PROGRAM S_Master_SMAC
VAR	 
eState								: E_SmacState;
	
/////////////////////////////////////////////INITIALIZATION FUNCTION/////////////////////////////////////////////////////
	fbSmacInitialization_L							: FB_SmacInitialization;
	I_O_fbSmacInitialization_L						:ST_Phasing_Home;

	fbSmacInitialization_R							: FB_SmacInitialization;
	I_O_fbSmacInitialization_R						:ST_Phasing_Home;

/////////////////////////////////////////////CYCLE/MANUAL FUNCTION/////////////////////////////////////////////////////
	fbSmacCycleMan									: FB_SmacCycleMan;
	bTest											: BOOL;
/////////////////////////////////////////////CTRL SMAC/////////////////////////////////////////////////////
	nHomeState										: DINT;	
	nCyclePickState									: DINT;
	nCycleScrewkState								: DINT;
	nHomeStateManual								: DINT;	
	nCyclePickStateManual							: DINT;
	nCycleScrewkStateManual							: DINT;
	bLinealHomed									: BOOL;
	bRotativeHomed									: BOOL;
	bFirstCycle										: BOOL;
	
	
	aCycleFlag										: ARRAY[0..10] OF BOOL;

/////////////////////////////////////////////ERROR FUNCTION/////////////////////////////////////////////////////	
	fbErrorRST										: FB_ErrorReset;
	bEnbale_ErrorRST								: BOOL;
	bResetErrors									: BOOL;
	bAllErrorsCleared								: BOOL;
/////////////////////////////////////////////TIMERS / TRIGGERS/////////////////////////////////////////////////////
	tonResetError									:Tc2_Standard.TON;
	tonAbortModule									:Tc2_Standard.TON;
	tonCaseDelay									: ARRAY[0..40] OF TON;
	rTrigCase										: ARRAY[0..10] OF R_TRIG;
	CMDTrig											: ARRAY[0..10] OF R_TRIG;										
/////////////////////////////////////////////GRIPPERS CONTROL/////////////////////////////////////////////////////
	bCatchPiece							:BOOL;	//If set to TRUE - gripper OPEN || FALSE - gripper CLOSED
	bGuideScrew							:BOOL;	//If set to TRUE - gripper OPEN || FALSE - gripper CLOSED
	bGripperGuide_Timeout				:BOOL;	//Gripper didn't close in 3sec
	bGripperFixture_Timeout				:BOOL;	//Gripper didn't close in 3sec
	fbGripper_Guide						:FB_GripperCtrl;	
	fbGripper_Fixture					:FB_GripperCtrl;

END_VAR//---------------------------------------------------------------------------------------oldschoo1
VAR_OUTPUT
	stSmacReport						:ST_ProcessReport;
END_VAR

//--------------------IN/OUT----------------------------------------*
VAR_INPUT
	bCloseGripper						: BOOL;
	CMD									:ST_ModuleCMD;	
END_VAR
VAR_OUTPUT
	STATUS								:ST_ModuleStatus;
	I_O_fbSmacCycleMan					: ST_CYC_MAN;
END_VAR




//----------------------------------------------------------oldschoo1

PRG_Fault_SMAC(aAlarms := GVL_Master.stAlarms);
b_Ctrl_Smac();
c_FunctionProcess();
d_TimTrig();

ACTION a_StringDefinitions:

//////////////////////////////////////////STATUS STRING DEFINITIONS/////////////////////////////////////////////////////

	stSmacIO.sStatus[0]:='Initialization done';
	stSmacIO.sStatus[1]:='Servo enabled';
	stSmacIO.sStatus[2]:='';
	stSmacIO.sStatus[3]:='Motion execution acknowledge bit';
	stSmacIO.sStatus[4]:='Trajectory complete';
	stSmacIO.sStatus[5]:='';
	stSmacIO.sStatus[6]:='Homing Success';
	stSmacIO.sStatus[7]:='Homing failure';
	stSmacIO.sStatus[8]:='Phasing Succes';
	stSmacIO.sStatus[9]:='Phasing failure';
	stSmacIO.sStatus[10]:='Macro execution error';
	stSmacIO.sStatus[11]:='Macro execution';
	stSmacIO.sStatus[12]:='General fault';
	stSmacIO.sStatus[13]:='Servo error';
	stSmacIO.sStatus[14]:='STO fault';
	stSmacIO.sStatus[15]:='STO status';
	stSmacIO.sStatus[16]:='STO Input 1 de-energized';
	stSmacIO.sStatus[17]:='STO Input 2 de-energized';
	stSmacIO.sStatus[18]:='I2T fault';
	stSmacIO.sStatus[19]:='Driver overtemperature fault';
	stSmacIO.sStatus[20]:='Initialization done';
	
//////////////////////////////////////////MODE OF OPERATION STRING DEFINITIONS/////////////////////////////////////////////////////
	
	stSmacIO.sModeOfOperation[0] :='';
	stSmacIO.sModeOfOperation[1] :='Absolute position move';
	stSmacIO.sModeOfOperation[2] :='Relative position move';
	stSmacIO.sModeOfOperation[3] :='Velocity move';
	stSmacIO.sModeOfOperation[4] :='Torque move';
	stSmacIO.sModeOfOperation[5] :='Current move/QM1';
	stSmacIO.sModeOfOperation[6] :='Homing';
	stSmacIO.sModeOfOperation[7] :='Phasing';
	stSmacIO.sModeOfOperation[8] :='Current move/QM2';
	stSmacIO.sModeOfOperation[9] :='';
	stSmacIO.sModeOfOperation[10] :='Macro execution**';
	
//////////////////////////////////////////CONTRO WORD STRING DEFINITIONS/////////////////////////////////////////////////////

stSmacIO.sControlWord[0] :='';
stSmacIO.sControlWord[1] :='Start motion/macro start';
stSmacIO.sControlWord[2] :='Stop motion';
stSmacIO.sControlWord[3] :='Motor off';
stSmacIO.sControlWord[4] :='Motor on';
stSmacIO.sControlWord[5] :='Fault reset';
END_ACTION

ACTION b_Ctrl_Smac:

IF cmd.bAbort OR NOT stSafety.bSafety_OK OR NOT cmd.bEnable   THEN
	eState									:= E_SmacState.ABORTED;
END_IF

IF CMDTrig[4].Q THEN
	eState									:= E_SmacState.RESET_ERROR;
END_IF

IF eState = E_SmacState.MANUAL THEN
	I_O_fbSmacCycleMan.bManual_fbSmacCycleMan := TRUE;
ELSE I_O_fbSmacCycleMan.bManual_fbSmacCycleMan := FALSE;
END_IF

IF CMD.bManualMode THEN
	eState									:= E_SmacState.MANUAL;
END_IF
									

CMDTrig[0]( CLK := cmd.bAbort OR NOT stSafety.bSafety_OK OR NOT cmd.bEnable );
CMDTrig[1]( CLK := CMD.bEnable AND tonCaseDelay[3].Q );
CMDTrig[2]( CLK := CMD.bExecute);
CMDTrig[3]( CLK := CMD.bManualMode);
CMDTrig[4]( CLK := CMD.bReset);

		
(*******************************************************CTRL***********************************************************)
// Axis CTRL State Machine
CASE eState OF //--------------------------------------------------------------------------------------------------SM
	
E_SmacState.ABORTED://-------------------------------------------------------------------------------------------ABORTED:

						IF tonCaseDelay[22].Q THEN
							eState 												:= E_SmacState.ERROR;						
						END_IF

						IF  CMD.bEnable THEN
							eState 												:= E_SmacState.HOMING;
						END_IF
						//RESETTING
						I_O_fbSmacInitialization_R.bFunctionRequest				:= FALSE;
						I_O_fbSmacInitialization_L.bFunctionRequest				:= FALSE;
						I_O_fbSmacInitialization_R.bReset						:= TRUE;
						I_O_fbSmacInitialization_L.bReset						:= TRUE;
						I_O_fbSmacInitialization_L.bAcknowledge					:= FALSE;
						I_O_fbSmacInitialization_R.bAcknowledge					:= FALSE;
						
						I_O_fbSmacCycleMan.bAutoCycleRequest					:= FALSE;
						I_O_fbSmacCycleMan.bResetAutoCycle						:= TRUE;
						I_O_fbSmacCycleMan.bInitSecondPart						:= FALSE;
						I_O_fbSmacCycleMan.bAutoCycleAcknowledge				:= FALSE;
						aCycleFlag[1]											:= FALSE;
						aCycleFlag[2]											:= FALSE;
						aCycleFlag[3]											:= FALSE;
						
						nHomeState												:= 0;
						nCyclePickState											:= 0;
						nCycleScrewkState										:= 0;
						
						bCloseGripper											:= FALSE;
						
						IF tonCaseDelay[3].Q THEN
							I_O_fbSmacInitialization_R.bReset					:= FALSE;
							I_O_fbSmacInitialization_L.bReset					:= FALSE;
							I_O_fbSmacInitialization_R.bEnable					:= FALSE;
							I_O_fbSmacInitialization_L.bEnable					:= FALSE;
							
							I_O_fbSmacCycleMan.bResetAutoCycle					:= FALSE;
							I_O_fbSmacCycleMan.bCycProcess						:= FALSE;
							
							I_O_fbSmacCycleMan.bResetAutoCycle					:= FALSE;
							I_O_fbSmacCycleMan.bCycProcess						:= FALSE;
						END_IF
						

E_SmacState.HOMING://---------------------------------------------------------------------------------------------HOMING:
////////////////////////////////////////////////////LINEAL HOME////////////////////////////////////////////////////
						CASE 	nHomeState	OF
								
						0:
						IF aCycleFlag[1] THEN
							eState 												:= E_SmacState.AXIS_READY;
						ELSE nHomeState											:= 200;
						END_IF
						200:
						I_O_fbSmacInitialization_L.bEnable						:= TRUE;
						IF tonCaseDelay[6].Q THEN
							nHomeState											:= 300;
						END_IF
						300:
						I_O_fbSmacInitialization_L.bFunctionRequest				:= TRUE;
						IF tonCaseDelay[7].Q THEN
							nHomeState											:= 400;
						END_IF
						400:
						IF I_O_fbSmacInitialization_L.bAcknowledgeRequest THEN
							I_O_fbSmacInitialization_L.bAcknowledge				:= TRUE;
							nHomeState											:= 500;
							bLinealHomed										:= TRUE;
						ELSIF I_O_fbSmacInitialization_L.bPhasingError OR I_O_fbSmacInitialization_L.bHomeError THEN
							nHomeState											:= 500;
						END_IF
						500:
						I_O_fbSmacInitialization_L.bReset						:= TRUE;
						IF tonCaseDelay[8].Q THEN
							nHomeState											:= 600;
						END_IF
						600:
						I_O_fbSmacInitialization_L.bEnable						:= FALSE;
						I_O_fbSmacInitialization_L.bReset						:= FALSE;
						I_O_fbSmacInitialization_L.bFunctionRequest				:= FALSE;
						I_O_fbSmacInitialization_L.bAcknowledge					:= FALSE;
						IF bLinealHomed THEN
							nHomeState											:= 1200;
						END_IF
						
						1200:
						I_O_fbSmacInitialization_R.bEnable						:= TRUE;
						IF tonCaseDelay[9].Q THEN
							nHomeState											:= 1300;
						END_IF
						1300:
						I_O_fbSmacInitialization_R.bFunctionRequest				:= TRUE;
						IF tonCaseDelay[10].Q THEN
							nHomeState											:= 1400;
						END_IF
						1400:
						IF I_O_fbSmacInitialization_R.bAcknowledgeRequest THEN
							I_O_fbSmacInitialization_R.bAcknowledge				:= TRUE;
							nHomeState											:= 1500;
							bRotativeHomed										:= TRUE;
						ELSIF I_O_fbSmacInitialization_R.bPhasingError OR I_O_fbSmacInitialization_R.bHomeError THEN
							nHomeState											:= 1500;
						END_IF
						1500:
						I_O_fbSmacInitialization_R.bReset						:= TRUE;
						IF tonCaseDelay[11].Q THEN
							nHomeState											:= 1600;
						END_IF
						1600:
						I_O_fbSmacInitialization_R.bEnable						:= FALSE;
						I_O_fbSmacInitialization_R.bReset						:= FALSE;
						I_O_fbSmacInitialization_R.bFunctionRequest				:= FALSE;
						I_O_fbSmacInitialization_R.bAcknowledge					:= FALSE;
						IF bRotativeHomed AND bLinealHomed THEN
							bRotativeHomed										:= FALSE;
							bLinealHomed										:= FALSE;
							aCycleFlag[1]										:= TRUE;
							nHomeState											:= 0;
						END_IF
						
						5000://ERROR

						IF tonCaseDelay[12].Q THEN
							eState 												:= E_SmacState.ABORTED;
						END_IF
						END_CASE
	
						IF I_O_fbSmacInitialization_R.bHomeError OR I_O_fbSmacInitialization_R.bPhasingError OR
							I_O_fbSmacInitialization_L.bHomeError OR I_O_fbSmacInitialization_L.bPhasingError OR CMDTrig[0].Q THEN
							nHomeState											:= 5000;
						END_IF

		
E_SmacState.AXIS_READY://-------------------------------------------------------------------------------------AXIS_READY:
							
							aCycleFlag[1]										:= FALSE;
							aCycleFlag[3]										:= FALSE;
							//GO TO FIRST PART OF THE CYCLE
							IF (CMDTrig[2].Q AND stSmac.bSet_PickScrew) OR rTrigCase[1].Q THEN
									eState := E_SmacState.Cycle_Pick_Part;
							END_IF
										
							
E_SmacState.Cycle_Pick_Part://---------------------------------------------------------------------------Cycle_Pick_Part:		
							CASE nCyclePickState OF
							0:
							IF aCycleFlag[2] THEN
							eState 												:= E_SmacState.Cycle_Screw;
							ELSE nCyclePickState								:= 200;
							END_IF
							200:
							IF NOT bFirstCycle THEN
								nCyclePickState									:= 300;
							ELSE nCyclePickState								:= 400;
							END_IF
							300:
							I_O_fbSmacCycleMan.bSetValues						:= TRUE;
							IF tonCaseDelay[15].Q THEN
								nCyclePickState									:= 400;
							END_IF
							400:
							I_O_fbSmacCycleMan.bCycProcess						:= TRUE;
							IF tonCaseDelay[16].Q THEN
								nCyclePickState									:= 500;
							END_IF
							500:
							I_O_fbSmacCycleMan.bAutoCycleRequest				:= TRUE; 
							IF tonCaseDelay[17].Q THEN
								nCyclePickState									:= 600;
							END_IF
							600:
							IF I_O_fbSmacCycleMan.bFirstPartDoneFlag THEN
								aCycleFlag[2]									:= TRUE;
								nCyclePickState									:= 0;
							END_IF
							
							5000://ERROR
							IF tonCaseDelay[18].Q THEN
								eState 											:= E_SmacState.ABORTED;
							END_IF
							END_CASE
	
							IF I_O_fbSmacCycleMan.bCycError  THEN
								nCyclePickState										:= 5000;
							END_IF

						
							
							
E_SmacState.Cycle_Screw://-----------------------------------------------------------------------------------Cycle_Screw:
							aCycleFlag[2]										:= FALSE;
							CASE nCycleScrewkState OF
							0:	
							IF aCycleFlag[3] THEN//second part request
								eState 											:= E_SmacState.RECORD_CYCLE_DATA;
							ELSE nCycleScrewkState								:= 100;
							END_IF
							100:
							IF I_O_fbSmacCycleMan.bFirstPartDoneFlag AND CMDTrig[2].Q AND stSmac.bSet_ScrewItIn THEN
								I_O_fbSmacCycleMan.bInitSecondPart				:= TRUE;
								nCycleScrewkState								:= 200;
							END_IF
							200:
							bCloseGripper									:= I_O_fbSmacCycleMan.bOpenGuideGripper;
							IF I_O_fbSmacCycleMan.bAutoCycleAcknowledgeRequest THEN
								I_O_fbSmacCycleMan.bAutoCycleAcknowledge		:= TRUE;
								nCycleScrewkState								:= 300;
								
							END_IF
							300:
							IF I_O_fbSmacCycleMan.bCycleProcessDone THEN
								nCycleScrewkState								:= 400;
								I_O_fbSmacCycleMan.bAutoCycleAcknowledge		:= FALSE;
								I_O_fbSmacCycleMan.bAutoCycleRequest			:= FALSE;
								I_O_fbSmacCycleMan.bInitSecondPart				:= FALSE;
								I_O_fbSmacCycleMan.bSetValues					:= FALSE;
								I_O_fbSmacCycleMan.bResetAutoCycle				:= TRUE;
								nCycleScrewkState								:= 400;
							END_IF 
							400:
							IF tonCaseDelay[18].Q THEN
								I_O_fbSmacCycleMan.bResetAutoCycle				:= FALSE;
								I_O_fbSmacCycleMan.bCycProcess					:= FALSE;
								nCycleScrewkState								:= 500;
							END_IF
							500:
							nCycleScrewkState									:= 0;
							aCycleFlag[3]										:= TRUE;
							
							5000://ERROR
							IF tonCaseDelay[18].Q THEN
								eState 											:= E_SmacState.ABORTED;
							END_IF
							END_CASE
	
							IF I_O_fbSmacCycleMan.bCycError THEN
								nCycleScrewkState								:= 5000;
							END_IF

E_SmacState.RECORD_CYCLE_DATA://-----------------------------------------------------------------------------RECORD_CYCLE_DATA:

							
							stSmacReport.rSmac_Settings_LinearAcc				:= I_O_fbSmacCycleMan.nScaledLinearAcc;
							stSmacReport.rSmac_Settings_LinearVel				:= I_O_fbSmacCycleMan.nScaledLinearVel;
							stSmacReport.rSmac_Settings_LinearTorque			:= I_O_fbSmacCycleMan.nScaledLinearTorque;
							stSmacReport.rSmac_Settings_RotativeAcc				:= I_O_fbSmacCycleMan.nScaledRotativeAcc;
							stSmacReport.rSmac_Settings_RotativeVel				:= I_O_fbSmacCycleMan.nScaledRotativeVel;
							
							stSmacReport.bSmac_Pass								:= I_O_fbSmacCycleMan.bPass;
							stSmacReport.bSmac_Fail								:= I_O_fbSmacCycleMan.bFail;
				
							stSmacReport.rSmac_MaxDistanceReached				:= I_O_fbSmacCycleMan.MaxDistanceReached;
							IF tonCaseDelay[13].Q THEN
								eState 											:= E_SmacState.AXIS_READY;
 							END_IF
							

E_SmacState.RESET_ERROR://-----------------------------------------------------------------------------------------------ERROR:
							IF bAllErrorsCleared AND tonCaseDelay[4].Q THEN
								bEnbale_ErrorRST								:= FALSE;
							ELSE bEnbale_ErrorRST								:= TRUE;
							END_IF
							IF bFlash1Hz AND bEnbale_ErrorRST THEN
								bResetErrors									:= TRUE;
							ELSE bResetErrors									:= FALSE;
							END_IF
							IF tonCaseDelay[5].Q AND tonCaseDelay[4].Q THEN
								eState := E_SmacState.ABORTED;
							END_IF

E_SmacState.MANUAL://---------------------------------------------------------------------------------------------------MANUAL:
							IF NOT CMD.bManualMode THEN
								eState := E_SmacState.ABORTED;
							END_IF
							
ELSE 
eState := E_AxisState.ABORTED;
END_CASE //------------------------------------------------------------------------------------------------------END_CASE

(******************************************************STATUS************************************************************)
// Module Status
status.bReady					:= eState = E_SmacState.AXIS_READY;

status.bBusy					:= 	eState = E_SmacState.Cycle_Screw	OR
				   					eState = E_SmacState.Cycle_Pick_Part OR
				   					eState = E_SmacState.HOMING;
status.bFirstPartOfCycleDone	:=	I_O_fbSmacCycleMan.bFirstPartDoneFlag;	
		   
status.bDone					:= 	eState =	E_SmacState.RECORD_CYCLE_DATA;

status.bError					:= 	I_O_fbSmacInitialization_L.bHomeError OR I_O_fbSmacInitialization_R.bHomeError OR
								I_O_fbSmacInitialization_L.bPhasingError OR I_O_fbSmacInitialization_R.bPhasingError OR
								I_O_fbSmacCycleMan.bCycError OR stSmacIO.inStatusWordRotative.13 OR stSmacIO.inStatusWordLinear.13  ;
//--------------------------------------------------GRIPPERS-------------------------------------------------------------oldschoo1

IF CMD_Smac.bFixtureGripper OR (I_O_fbSmacCycleMan.bCloseFixtureGripper AND eState = E_AxisState.MANUAL_MODE) THEN
	bCatchPiece					:= TRUE;
ELSE bCatchPiece					:= FALSE;
END_IF

IF (CMD_Smac.bGuideGripper AND NOT bCloseGripper ) OR 
	(I_O_fbSmacCycleMan.bCloseGuideGripper AND eState = E_AxisState.MANUAL_MODE)THEN
	bGuideScrew					:= TRUE;
ELSE bGuideScrew					:= FALSE;
END_IF
END_ACTION

ACTION c_FunctionProcess:
//LINEAR PHASING AND HOME
fbSmacInitialization_L(	//INPUTS:
						bEnable 				:= I_O_fbSmacInitialization_L.bEnable,
						bAcknowledge 			:= I_O_fbSmacInitialization_L.bAcknowledge,
						bReset					:= I_O_fbSmacInitialization_L.bReset,
						bFunctionRequest		:= I_O_fbSmacInitialization_L.bFunctionRequest,
						nStatusWord				:= stSmacIO.inStatusWordLinear,
						nCurrentModeOfOperation	:= stSmacIO.inModeOfOperationLinear,							
						
						//OUTPUTS	
						bFunctionEnabled		=> I_O_fbSmacInitialization_L.bFunctionEnabled,
						bPhasingProcessDone		=> I_O_fbSmacInitialization_L.bPhasingProcessDone,
						bHomingProcessDone		=> I_O_fbSmacInitialization_L.bHomingProcessDone,
						bAcknowledgeRequest		=> I_O_fbSmacInitialization_L.bAcknowledgeRequest,
						bHomeError				=> I_O_fbSmacInitialization_L.bHomeError,
						bPhasingError			=> I_O_fbSmacInitialization_L.bPhasingError,
						//IN/OUT
						nControlWord			:= stSmacIO.qnControlWordLinear,								
						nModeOfOperation		:= stSmacIO.qnModeOfOperationLinear);
						
//ROTATIVE PHASING AND HOME						
fbSmacInitialization_R(	//INPUTS:
						bEnable 				:= I_O_fbSmacInitialization_R.bEnable,
						bAcknowledge 			:= I_O_fbSmacInitialization_R.bAcknowledge,
						bReset					:= I_O_fbSmacInitialization_R.bReset,
						bFunctionRequest		:= I_O_fbSmacInitialization_R.bFunctionRequest,
						nStatusWord				:= stSmacIO.inStatusWordRotative,
						nCurrentModeOfOperation	:= stSmacIO.inModeOfOperationRotative,							
						
						//OUTPUTS	
						bFunctionEnabled		=> I_O_fbSmacInitialization_R.bFunctionEnabled,
						bPhasingProcessDone		=> I_O_fbSmacInitialization_R.bPhasingProcessDone,
						bHomingProcessDone		=> I_O_fbSmacInitialization_R.bHomingProcessDone,
						bAcknowledgeRequest		=> I_O_fbSmacInitialization_R.bAcknowledgeRequest,
						bHomeError				=> I_O_fbSmacInitialization_R.bHomeError,
						bPhasingError			=> I_O_fbSmacInitialization_R.bPhasingError,
						//IN/OUT
						nControlWord			:= stSmacIO.qnControlWordRotative,								
						nModeOfOperation		:= stSmacIO.qnModeOfOperationRotative);
//CYCLE / MANUAL						
fbSmacCycleMan(			//INPUTS:
						nLinearVel				:= I_O_fbSmacCycleMan.nLinearVel,
						nLinearAcc				:= I_O_fbSmacCycleMan.nLinearAcc,
						nLinearSetPoint			:= I_O_fbSmacCycleMan.nLinearSetPoint,
						nLinearTorque			:= I_O_fbSmacCycleMan.nLinearTorque,
						bRotativeWorkPosition	:= I_O_fbSmacCycleMan.nRotativeWorkPosition,
						
						nRotativeVel			:= I_O_fbSmacCycleMan.nRotativeVel,
						nRotativeAcc			:= I_O_fbSmacCycleMan.nRotativeAcc,
						nRotativeSetPoint		:=  GVL_PERSISTENT.nSmacRotativeSetPoint,
						
						bCycProcess				:= I_O_fbSmacCycleMan.bCycProcess,
						bAutoCycleAcknowledge	:= I_O_fbSmacCycleMan.bAutoCycleAcknowledge,
						bAutoCycleRequest		:= I_O_fbSmacCycleMan.bAutoCycleRequest,
						bResetAutoCycle			:= I_O_fbSmacCycleMan.bResetAutoCycle,
						bInitSecondPart			:= I_O_fbSmacCycleMan.bInitSecondPart,
						bSetValues				:= GVL_HMI.bSmacSetValue OR (NOT bFirstCycle AND I_O_fbSmacCycleMan.bSetValues),
						bFixtureGripperClosed	:= stSmac.bGripperB_ClosedSensor,
						bGuideGripperClosed		:= stSmac.bGripperA_ClosedSensor,
						bManual					:= I_O_fbSmacCycleMan.bManual_fbSmacCycleMan,
						
						nDistanceSetPoint		:= I_O_fbSmacCycleMan.nDistanceSetPoint,				
						nDistanceTolerance		:= 500, //I_O_fbSmacCycleMan.nDistanceTolerance,
						bPickCycleMan			:= GVL_HMI.bSmacCyc1,
						bScrewCycleMan			:= GVL_HMI.bSmacCyc2,
						bHomeMan				:= GVL_HMI.bSmacHOME,
						//OUTPUTS
						bAutoCycleAcknowledgeRequest 	=> I_O_fbSmacCycleMan.bAutoCycleAcknowledgeRequest,
						bCycleProcessDone				=> I_O_fbSmacCycleMan.bCycleProcessDone,
						bFirstPartDoneFlag				=> I_O_fbSmacCycleMan.bFirstPartDoneFlag,
						bCycError						=> I_O_fbSmacCycleMan.bCycError,
						bOpenGuideGripper				=> I_O_fbSmacCycleMan.bOpenGuideGripper,
						bCloseGuideGripper				=> I_O_fbSmacCycleMan.bCloseGuideGripper,
						bCloseFixtureGripper			=> I_O_fbSmacCycleMan.bCloseFixtureGripper,
						bPass							=> I_O_fbSmacCycleMan.bPass,										
						bFail							=> I_O_fbSmacCycleMan.bFail,
						
						nScaledLinearVel				=> I_O_fbSmacCycleMan.nScaledLinearVel,			
						nScaledLinearAcc				=> I_O_fbSmacCycleMan.nScaledLinearAcc,						
						nScaledLinearSetPoint			=> I_O_fbSmacCycleMan.nScaledLinearSetPoint,						
						nScaledLinearTorque				=> I_O_fbSmacCycleMan.nScaledLinearTorque,					
	
						nScaledRotativeVel				=> I_O_fbSmacCycleMan.nScaledRotativeVel,						
						nScaledRotativeAcc				=> I_O_fbSmacCycleMan.nScaledRotativeAcc,					
						nScaledRotativeSetPoint			=> I_O_fbSmacCycleMan.nScaledRotativeSetPoint,
						MaxDistanceReached				=> I_O_fbSmacCycleMan.MaxDistanceReached,	
						bScrewAnimation					=> GVL_HMI.bScrewAnimation,
						//IN/OUT
						stSmacIO				:= stSmacIO);
						
							
									
												
//ERROR RESET
fbErrorRST(				//INPUTS
						bEnbale					:= bEnbale_ErrorRST,
						bResetErrors			:= bResetErrors,
						//OUTPUTS
						bAllErrorsCleared		=> bAllErrorsCleared,
						//IN/OUT
						stSmacIO				:= stSmacIO,
						bHomeError_L			:= I_O_fbSmacInitialization_L.bHomeError,
						bHomeError_R			:= I_O_fbSmacInitialization_R.bHomeError,
						bPhasingError_L			:= I_O_fbSmacInitialization_L.bPhasingError,
						bPhasingError_R			:= I_O_fbSmacInitialization_R.bPhasingError,
						bCycleError				:= I_O_fbSmacCycleMan.bCycError);

// Grippers CTRL
fbGripper_Fixture	 (bCloseGrip		:=bCatchPiece,
					  bClosedSensor		:=stSmac.bGripperB_ClosedSensor,
					  bOpen_Sig			=>stSmac.bGripperB_Open,
					  bClose_Sig		=>stSmac.bGripperB_Close,
					  bTimeout			=>bGripperFixture_Timeout);


fbGripper_Guide	     (bCloseGrip		:=bGuideScrew,
					  bClosedSensor		:=stSmac.bGripperA_ClosedSensor,
					  bOpen_Sig			=>(stSmac.bGripperA_Open ),
					  bClose_Sig		=>stSmac.bGripperA_Close,
					  bTimeout			=>bGripperGuide_Timeout);
END_ACTION

ACTION d_TimTrig:
//TIMERS

tonCaseDelay[0](IN := (eState =E_SmacState.HOMING) , PT := T#1S);
tonCaseDelay[1(*10*)](IN := eState = E_SmacState.Cycle_Screw , PT := T#1S);
tonCaseDelay[16](IN := eState = E_SmacState.Cycle_Pick_Part , PT := T#500MS);
tonCaseDelay[3](IN := (eState = E_SmacState.ABORTED) , PT := T#1S);
tonCaseDelay[4](IN := eState = E_SmacState.ERROR , PT := T#1S);
tonCaseDelay[13](IN := eState = E_SmacState.RECORD_CYCLE_DATA , PT := T#500MS);


tonCaseDelay[5](IN :=bAllErrorsCleared , PT := T#500MS);
tonCaseDelay[6](IN := nHomeState = 200 , PT := T#500MS);
tonCaseDelay[7](IN := nHomeState = 300 , PT := T#500MS);
tonCaseDelay[8](IN := nHomeState = 500 , PT := T#500MS);
tonCaseDelay[9](IN := nHomeState = 1200 , PT := T#500MS);
tonCaseDelay[10](IN := nHomeState = 1300 , PT := T#500MS);
tonCaseDelay[11](IN := nHomeState = 1500 , PT := T#500MS);
tonCaseDelay[12](IN := nHomeState = 5000 , PT := T#2S);

tonCaseDelay[15](IN := nCyclePickState = 300 , PT := T#500MS);
tonCaseDelay[16](IN := nCyclePickState = 400 , PT := T#500MS);  //??? the Same line 5
tonCaseDelay[17](IN := nCyclePickState = 500 , PT := T#500MS);
tonCaseDelay[18](IN := nCycleScrewkState = 400 , PT := T#500MS);


tonCaseDelay[21](IN := (stSmacIO.qnControlWordLinear = 2) , PT := T#1S);
tonCaseDelay[22](IN :=  stSmacIO.inStatusWordRotative.15 OR stSmacIO.inStatusWordRotative.16 OR
						 stSmacIO.inStatusWordRotative.17 OR stSmacIO.inStatusWordLinear.15 OR
						 stSmacIO.inStatusWordLinear.16 OR stSmacIO.inStatusWordLinear.17 
						, PT := T#500MS);

tonCaseDelay[23](IN :=cmd.bAbort OR NOT stSafety.bSafety_OK OR NOT cmd.bEnable , PT := T#1S);
tonCaseDelay[24](IN :=I_O_fbSmacCycleMan.bCycleProcessDone , PT := T#3S);


tonCaseDelay[26](IN := nHomeStatemanual = 200 , PT := T#500MS);
tonCaseDelay[27](IN := nHomeStatemanual = 300 , PT := T#500MS);
tonCaseDelay[28](IN := nHomeStatemanual = 500 , PT := T#500MS);
tonCaseDelay[29](IN := nHomeStatemanual = 1200 , PT := T#500MS);
tonCaseDelay[30](IN := nHomeStatemanual = 1300 , PT := T#500MS);
tonCaseDelay[31](IN := nHomeStatemanual = 1500 , PT := T#500MS);
tonCaseDelay[32](IN := nHomeStatemanual = 5000 , PT := T#2S);

tonCaseDelay[35](IN := nCyclePickStatemanual = 300 , PT := T#500MS);
tonCaseDelay[36](IN := nCyclePickStatemanual = 400 , PT := T#500MS);  //??? the Same line 5
tonCaseDelay[37](IN := nCyclePickStatemanual = 500 , PT := T#500MS);
tonCaseDelay[38](IN := nCycleScrewkStatemanual = 400 , PT := T#500MS);


//TRIGGERS
rTrigCase[0](CLK := eState = E_SmacState.ABORTED);
END_ACTION

END_PROGRAM

(* stored: Version 1.1.0.1, ProductVersion 3.1.4024.12
   POU S_Master_SMAC: Id {e9c13e85-b7ea-4c18-8786-d25414b50222}, SpecialFunc None
   Action a_StringDefinitions: Id {d280c89d-ed1a-4069-a1bc-5559c561d7d0}
   Action b_Ctrl_Smac: Id {ed1ca0da-bb44-4a29-9b4f-e40d75958aab}
   Action c_FunctionProcess: Id {cb31e280-c9f0-495e-8973-5eb73320880b}
   Action d_TimTrig: Id {c5245bf9-327c-4c9a-83c0-3a10a0300d92} *)
